(* IEC 61131-3 sources: ELE33052024DA/src/OpenPLC/build, 2 files *)

(* ---- plc.st ---- *)
TYPE
  LOGLEVEL : (CRITICAL, WARNING, INFO, DEBUG) := INFO;
END_TYPE

FUNCTION_BLOCK LOGGER
  VAR_INPUT
    TRIG : BOOL;
    MSG : STRING;
    LEVEL : LOGLEVEL := INFO;
  END_VAR
  VAR
    TRIG0 : BOOL;
  END_VAR

  IF TRIG AND NOT TRIG0 THEN
  {{
   LogMessage(GetFbVar(LEVEL),(char*)GetFbVar(MSG, .body),GetFbVar(MSG, .len));
  }}
  END_IF;
  TRIG0:=TRIG;
END_FUNCTION_BLOCK

PROGRAM aqua_sys
  VAR
    low_DO : BOOL;
    high_DO : BOOL;
    airpump : BOOL;
    pH : BOOL;
    pHalert : BOOL;
    low_temp : BOOL;
    high_temp : BOOL;
    heating : BOOL;
    waterpump : BOOL;
    wp_on : BOOL;
    wp_off : BOOL;
    wplatched : BOOL;
  END_VAR

  airpump := NOT(high_DO) AND (airpump OR low_DO);
  pHalert := pH;
  heating := low_temp;
  waterpump := NOT(low_temp) AND (high_temp OR wplatched);
  wplatched := NOT(wp_off) AND (wp_on OR wplatched);
END_PROGRAM

CONFIGURATION Config0

  RESOURCE Res0 ON PLC
    TASK task0(INTERVAL := T#20ms,PRIORITY := 0);
    PROGRAM instance0 WITH task0 : aqua_sys;
  END_RESOURCE
END_CONFIGURATION

(* ---- generated_plc.st ---- *)
PROGRAM aqua_sys
  VAR
    low_DO AT %QX0.0 : BOOL;
    high_DO AT %QX0.1 : BOOL;
    airpump AT %QX0.2 : BOOL;
    pH AT %QX0.3 : BOOL;
    pHalert AT %QX0.4 : BOOL;
    low_temp AT %QX0.5 : BOOL;
    high_temp AT %QX0.6 : BOOL;
    heating AT %QX0.7 : BOOL;
    waterpump AT %QX1.0 : BOOL;
    wp_on AT %QX1.1 : BOOL;
    wp_off AT %QX1.2 : BOOL;
    wplatched AT %QX1.3 : BOOL;
  END_VAR

  airpump := NOT(high_DO) AND (airpump OR low_DO);
  pHalert := pH;
  heating := low_temp;
  waterpump := NOT(low_temp) AND (high_temp OR wplatched);
  wplatched := NOT(wp_off) AND (wp_on OR wplatched);
END_PROGRAM

CONFIGURATION Config0

  RESOURCE Res0 ON PLC
    TASK task0(INTERVAL := T#20ms,PRIORITY := 0);
    PROGRAM instance0 WITH task0 : aqua_sys;
  END_RESOURCE
END_CONFIGURATION
